    path_answer = node_rpc_server.rqmovesinit(rq_moves_node_id)
    verify_path_answer(path_answer)

    approach_position_joints = get_inverse_kin(approach_pose, qnear=approach_joints)
    movej(approach_position_joints)

    node_rpc_server.movejdefinewaypoint(rq_movej_node_id, get_actual_joint_positions(), 1.0, 1.0)
    node_rpc_server.setparentid(rq_movej_node_id, move_force_node_id)
    reset_node_executor()
    active_and_reset_node(move_force_node_id)
    node_execution_thread = execute_node(rq_movej_node_id, True)

    path_answer = node_rpc_server.rqmovesinit(rq_moves_node_id)
    verify_path_answer(path_answer)
    q0 = node_rpc_server.rqmovesgetfirstpoint(rq_moves_node_id)
    node_rpc_server.setparentid(rq_movej_node_id, move_force_node_id)
    node_rpc_server.movejdefinewaypoint(rq_movej_node_id, q0, 1.0, 0.4)
    execute_node(rq_movej_node_id)
    execute_node(start_waypoint_node_id)
    execute_node(end_waypoint_node_id)

    kill_thread(node_execution_thread)

    node_rpc_server.movejdefinewaypoint(rq_movej_node_id, get_actual_joint_positions(), 1.0, 1.0)
    node_rpc_server.setparentid(rq_movej_node_id, contact_force_node_id)
    reset_node_executor()
    active_and_reset_node(contact_force_node_id)
    node_execution_thread = execute_node(rq_movej_node_id, True)

    timeout = 20
    while (point_dist(get_actual_tcp_pose(), stop_pose) > end_reached_threshold):
      if (timeout <= 0):
        popup("Door has not reached its final position")
        halt
      else:
        sync()
        timeout = timeout - get_steptime()
      end
    end

    kill_thread(node_execution_thread)

    approach_pose_in_start_frame = pose_trans(pose_inv(start_pose), approach_pose)
    retract_pose = pose_trans(get_actual_tcp_pose(), approach_pose_in_start_frame)
    movej(retract_pose)

    node_rpc_server.deletenode(move_force_node_id)
    node_rpc_server.deletenode(rq_moves_node_id)
    node_rpc_server.deletenode(start_waypoint_node_id)
    node_rpc_server.deletenode(end_waypoint_node_id)
    node_rpc_server.deletenode(contact_force_node_id)
    node_rpc_server.deletenode(rq_movej_node_id)

  end

  ###################################################################################
  #
  # CNC Insertion
  #
  ###################################################################################

  def rq_collet_insertion(contact_pose, insert_pose, inserted_pose):
      movel(contact_pose, a=1.2, v=0.025)
      movel(insert_pose, a=1.2, v=0.025)

      rq_ft_sensor_disconnected_check()
      rq_zero_sensor()
      sleep(0.1)

      direction = "Z+"
      stop_force_threshold = 3.0
      max_radius = 5.0
      radius_incr = 0.7
      peck_mode = False
      tangential_speed = 0.02
      compliant_insert_force_threshold = 10.0
      spiral_initial_pose_offset_name = "spiral_initial_pose_offset_name"
      rq_ins_destination = inserted_pose
      max_distance = point_dist(inserted_pose, get_actual_tcp_pose())
      rq_spiral_not_completed = False
      rq_ins_speed_setting = 0.02

      rq_insert_spiral_urcap(direction, stop_force_threshold, max_radius, radius_incr, peck_mode, tangential_speed, compliant_insert_force_threshold, spiral_initial_pose_offset_name)

      if (rq_spiral_not_completed):
        return False
      end

      return True
  end

  def rq_push_part(approach_pose, chuck_pose):
      rq_ft_sensor_disconnected_check()
      rq_zero_sensor()
      sleep(0.1)

      # Find pose with z axis pointing in the direction of the insertion
      p1 = translate_to_origin(approach_pose)
      insertion_dir_in_base_frame = pose_trans(p1, pose_trans(pose_inv(approach_pose), chuck_pose))
      ref_frame_pose = list_to_pose(kinematics_rpc_server.poseFromZaxis([insertion_dir_in_base_frame[0], insertion_dir_in_base_frame[1], insertion_dir_in_base_frame[2]]))

      surface_found = rq_linear_search_custom_frame("Z+", 10.0, 0.025, 0.1, ref_frame_pose)

      if not(surface_found):
          return False
      end

      return True
  end

  def rq_place_in_chuck(close_chuck_do, open_chuck_do, chuck_approach, chuck_position, chuck_delay):
      rq_open_workholding(close_chuck_do, open_chuck_do)

      movel(chuck_approach, a=1.2, v=0.25)
      movel(chuck_position, a=1.2, v=0.25)

      rq_close_workholding(close_chuck_do, open_chuck_do)
      sleep(chuck_delay)
  end

  def rq_pre_pick_in_chuck(chuck_approach, chuck_position, speed=0.25, accel=1.2):
      movel(chuck_approach, accel, speed)
      movel(chuck_position, accel, speed)
  end

  def rq_post_pick_in_chuck(close_chuck_do, open_chuck_do, chuck_approach, chuck_position, chuck_delay, speed=0.25,
  accel=1.2):
      rq_open_workholding(close_chuck_do, open_chuck_do)
      sleep(chuck_delay)

      movel(chuck_approach, accel, speed)
  end

  def rq_open_workholding(close_do, open_do):
      rq_set_workholding_do(close_do, open_do, False)
  end

  def rq_close_workholding(close_do, open_do):
      rq_set_workholding_do(close_do, open_do, True)
  end

  def rq_set_workholding_do(close_do, open_do, close_request):
      is_close_do_valid = rq_is_do_valid(close_do)
      is_open_do_valid = rq_is_do_valid(open_do)

      if(is_close_do_valid):
          set_standard_digital_out(close_do, close_request)
      end
      if(is_open_do_valid):
          set_standard_digital_out(open_do, not close_request)
      end
      if(is_close_do_valid or is_open_do_valid):
          sleep(0.5)
      end
  end

  def rq_is_do_valid(do_id):
      return do_id >= 0 and do_id <= 7
  end

  def set_cleaning_digital_output(address, state, blow_off_mode, output_type):
     if(blow_off_mode == BLOW_OFF_MODE_SMART_AIR):
       rq_set_output(output_type, address, state)
     end
  end

  ###################################################################################
  #
  # PATH GENERATOR 6 POINTS CURVE BUILT WITH 2 POINTS
  #
  ###################################################################################

  def execute_half_pipe(pose_1, pose_2,pose_transformation_air_nozzle_to_actual_tcp, depth, length_distance, width, angle, speed, spacing, address, output_type, blow_off_mode, passes):
    path_gen_poses = get_path_generator_6_points_poses(pose_1, pose_2, pose_transformation_air_nozzle_to_actual_tcp, depth, length_distance, width, angle)
    start_pose = p[path_gen_poses[0,0],path_gen_poses[0,1],path_gen_poses[0,2],path_gen_poses[0,3],path_gen_poses[0,4],path_gen_poses[0,5]]
    path_generator_node_id = setup_path_generator_6_points(path_gen_poses, speed, spacing)
    execute_path_generator_6_points(path_generator_node_id, start_pose,  address, output_type, blow_off_mode, passes)
  end

  def get_path_generator_6_points_poses(pose_2, pose_5,pose_transformation_air_nozzle_to_actual_tcp, depth=0.01, length=0, width=0.05, angle_deg=0):

    def offset_pose(pose, offset, offset_reference_frame, pose_transformation_air_nozzle_to_actual_tcp):
      pose_relative_to_ref_frame = express_pose_A_relative_to_pose_B(pose, offset_reference_frame)
      ref_frame_with_offset = pose_trans(offset_reference_frame, offset)
      pose_with_offset = pose_trans(ref_frame_with_offset, pose_relative_to_ref_frame)
      pose_with_offset_for_actual_tcp = pose_trans(pose_with_offset, pose_transformation_air_nozzle_to_actual_tcp)
      return pose_to_list(pose_with_offset_for_actual_tcp)
    end

    if(length > 0):
      middle_pose = interpolate_pose(pose_2, pose_5, 0.5)

      poses = get_symmetric_poses_from_middle(pose_2, pose_5, middle_pose, length)
      pose_2 = poses[0]
      pose_5 = poses[1]
    end

    path_ref_frame = list_to_pose(kinematics_rpc_server.reorientP1WithXTowardP2andZApproxP1Z(pose_2, pose_5))

    offset1 = pose_add(p[0,0,0,0,d2r(angle_deg),0], p[0, width,-depth,-d2r(angle_deg),0,0])
    offset2 = pose_add(p[0,0,0,0,d2r(angle_deg),0], p[0,     0,     0,              0,0,0])
    offset3 = pose_add(p[0,0,0,0,d2r(angle_deg),0], p[0,-width,-depth, d2r(angle_deg),0,0])

    pose_1_array = offset_pose(pose_2, offset1, path_ref_frame, pose_transformation_air_nozzle_to_actual_tcp)
    pose_2_array = offset_pose(pose_2, offset2, path_ref_frame, pose_transformation_air_nozzle_to_actual_tcp)
    pose_3_array = offset_pose(pose_2, offset3, path_ref_frame, pose_transformation_air_nozzle_to_actual_tcp)

    pose_4_array = offset_pose(pose_5, offset1, path_ref_frame, pose_transformation_air_nozzle_to_actual_tcp)
    pose_5_array = offset_pose(pose_5, offset2, path_ref_frame, pose_transformation_air_nozzle_to_actual_tcp)
    pose_6_array = offset_pose(pose_5, offset3, path_ref_frame, pose_transformation_air_nozzle_to_actual_tcp)

    return [pose_1_array, pose_2_array, pose_3_array, pose_4_array, pose_5_array, pose_6_array]
  end

  def setup_path_generator_6_points(pose_list, tcp_speed=0.1, spacing=0.02):

    def json_path_generator_node(pose_list, tcp_speed, spacing):

      SIX_POINTS_CURVE = 3
      OFFSET_TYPE_NONE = 0
      FORCE_OPPOSITE_SIDE = 2

      json = "{"
      json = concat(json, key_val("tcpSpeed", tcp_speed), ",")
      json = concat(json, key_val("poses", pose_list), ",")
      json = concat(json, key_val("avoidAbruptEnd", "false"), ",")
      json = concat(json, key_val("isSurfaceFillOn", "true"), ",")
      json = concat(json, key_val("spacing", spacing), ",")
      json = concat(json, key_val("pathType", SIX_POINTS_CURVE), ",")
      json = concat(json, key_val("offsetType",OFFSET_TYPE_NONE), ",")
      json = concat(json, key_val("endingMode", FORCE_OPPOSITE_SIDE), "}")

      return json
    end

    rq_path_generator_parent_id = 0
    path_generator_node_id = node_rpc_server.createPathGeneratorNode()
    node_rpc_server.fromjson(path_generator_node_id, json_path_generator_node(pose_list, tcp_speed, spacing))
    node_rpc_server.setparentid(path_generator_node_id, rq_path_generator_parent_id)

    return path_generator_node_id
  end

  def execute_path_generator_6_points(path_generator_node_id, pose_1, address = INVALID_OUTPUT_ADDRESS, output_type = MODBUS_TYPE, blow_off_mode = BLOW_OFF_MODE_NO_AIR, passes = 1):
    index = 0
    while (index < passes):
      movej(get_inverse_kin(pose_1))
      set_cleaning_digital_output(address, True, blow_off_mode, output_type)
      reset_node_executor()
      node_execution_thread = execute_node(path_generator_node_id, True)
      rq_continue_node_execution = False
      set_cleaning_digital_output(address, False, blow_off_mode, output_type)
      join node_execution_thread
      index = index + 1
    end
    node_rpc_server.deletenode(path_generator_node_id)
  end

  ###################################################################################
  #
  # Straight line trajectory
  #
  ###################################################################################

  def execute_straight_line(p1, p2,pose_transformation_air_nozzle_to_actual_tcp, accel=1.2, speed=0.25, distance = 0, angles = [0, 0, 0], address = INVALID_OUTPUT_ADDRESS, output_type = MODBUS_TYPE, blow_off_mode = BLOW_OFF_MODE_NO_AIR, passes = 1):
    offset_for_angles = p[0, 0, 0, d2r(angles[0]), d2r(angles[1]), d2r(angles[2])]
    p1 = pose_trans(p1, offset_for_angles)
    p2 = pose_trans(p2, offset_for_angles)

    # apply transformation to take into account that the actual tcp offset is not the same as the one that was used when the waypoints were saved:
    p1 = pose_trans(p1, pose_transformation_air_nozzle_to_actual_tcp)
    p2 = pose_trans(p2, pose_transformation_air_nozzle_to_actual_tcp)
    global air_output_adress = address

    qActual = get_actual_joint_positions()
    CleanPathId = node_rpc_server.createnewcleaningpathnode(p1, p2, qActual, passes, distance, accel, speed, blow_off_mode)

    reset_node_executor()
    if output_type == MODBUS_TYPE:
      air_thread = run modbusAirControlThread()
    elif output_type == STANDARD_TYPE:
      air_thread = run standardAirControlThread()
    end

    node_execution_thread = execute_node(CleanPathId, True)
    rq_continue_node_execution = False

    join node_execution_thread
    node_rpc_server.deletenode(CleanPathId)
    if output_type == MODBUS_TYPE or output_type == STANDARD_TYPE :
      kill air_thread
    end
  end

  ###################################################################################
  #
  # Cross trajectory
  #
  ###################################################################################

  def find_cross_trajectory_poses(p1, p2, height=0, width=0, p1_angles = [0, 0, 0], p2_angles = [0, 0, 0], p3_angles = [0, 0, 0], p4_angles = [0, 0, 0]):
    def find_side_poses(p0, p1):
      def find_side_pose(p0,p1,angle):
        p1_T_p0 = pose_trans(pose_inv(p0), p1)
        rotated_p0_by_90_degrees = pose_trans(p0, p[0, 0, 0, 0, 0, d2r(angle)])

        side_pose = pose_trans(rotated_p0_by_90_degrees, p1_T_p0)
        side_pose[3] = p0[3]
        side_pose[4] = p0[4]
        side_pose[5] = p0[5]

        return side_pose
      end

      p3= find_side_pose(p0, p1, 90)
      p4 = find_side_pose(p0, p1, 270)

      return [p3, p4]
    end

    def get_start_and_end_poses_based_on_distance(p1, p2, middle_pose, distance):
      if(distance == 0):
        start_pose = p1
        end_pose = p2
      else:
        poses = get_symmetric_poses_from_middle(p1, p2, middle_pose, distance)
        start_pose = poses[0]
        end_pose = poses[1]
      end
      return [start_pose, end_pose]
    end

    def get_side_poses_based_on_distance(p1, p2, middle_pose, width):
      if(width == 0):
        side_poses = find_side_poses(middle_pose, p1)
      else:
        poses = get_symmetric_poses_from_middle(p1, p2, middle_pose, width)
        side_poses = find_side_poses(middle_pose, poses[0])
      end

      return side_poses
    end

    def get_angle_offset(angles):
      return  p[0, 0, 0, d2r(angles[0]), d2r(angles[1]), d2r(angles[2])]
    end

    middle_pose = interpolate_pose(p1, p2, 0.5)

    start_and_end_poses = get_start_and_end_poses_based_on_distance(p1, p2, middle_pose, height)
    side_poses = get_side_poses_based_on_distance(p1, p2, middle_pose, width)

    p1_offset = get_angle_offset(p1_angles)
    p2_offset = get_angle_offset(p2_angles)
    p3_offset = get_angle_offset(p3_angles)
    p4_offset = get_angle_offset(p4_angles)

    start_and_end_poses[0] = pose_trans(start_and_end_poses[0], p1_offset)
    start_and_end_poses[1] = pose_trans(start_and_end_poses[1], p2_offset)
    side_poses[0] = pose_trans(side_poses[0], p3_offset)
    side_poses[1] = pose_trans(side_poses[1], p4_offset)

    return [middle_pose, start_and_end_poses[0], start_and_end_poses[1], side_poses[0], side_poses[1]]
  end

  def execute_cross_trajectory(p1, p2,pose_transformation_air_nozzle_to_actual_tcp, height=0, width=0, p1_angles = [0, 0, 0], p2_angles = [0, 0, 0], p3_angles = [0, 0, 0], p4_angles = [0, 0, 0], accel=1.2, speed=0.25,  address = INVALID_OUTPUT_ADDRESS, output_type = MODBUS_TYPE, blow_off_mode = BLOW_OFF_MODE_NO_AIR, passes = 1):

    cross_poses = find_cross_trajectory_poses(p1, p2, height, width, p1_angles, p2_angles, p3_angles, p4_angles)

    p0 = pose_trans(cross_poses[0], pose_transformation_air_nozzle_to_actual_tcp)
    p1 = pose_trans(cross_poses[1], pose_transformation_air_nozzle_to_actual_tcp)
    p2 = pose_trans(cross_poses[2], pose_transformation_air_nozzle_to_actual_tcp)
    p3 = pose_trans(cross_poses[3], pose_transformation_air_nozzle_to_actual_tcp)
    p4 = pose_trans(cross_poses[4], pose_transformation_air_nozzle_to_actual_tcp)

   index = 0

   while (index < passes):
     movej(get_inverse_kin(p0))
     set_cleaning_digital_output(address, True, blow_off_mode, output_type)
     movel(p1, accel, speed)
     movel(p2, accel, speed)
     movel(p0, accel, speed)
     movel(p3, accel, speed)
     movel(p4, accel, speed)
     set_cleaning_digital_output(address, False, blow_off_mode, output_type)
     index = index + 1
   end
  end

  def execute_waypoint_cross_trajectory(starting_pose, finishing_pose, accel=1.2, speed=0.25):
   movej(get_inverse_kin(starting_pose))
   movel(finishing_pose, accel, speed)
  end

  ###################################################################################
  #
  # Fermat spiral trajectory
  #
  ###################################################################################

  def execute_fermat_spiral(start_pose, end_pose,pose_transformation_air_nozzle_to_actual_tcp, max_radius = 0, angle = 0, number_of_turns = 1, speed = 0.25,address = INVALID_OUTPUT_ADDRESS, output_type = MODBUS_TYPE, blow_off_mode = BLOW_OFF_MODE_NO_AIR, passes = 1):
    def find_middle(start_pose, end_pose):
      alpha = 0.5
      return interpolate_pose(start_pose, end_pose, alpha)
    end

    def find_next_theta(spiral_constant, theta, speed):
      denom = spiral_constant * sqrt(1/(4*theta) + theta)
      theta_dot = speed / denom
      theta = theta + theta_dot * rq_controller_time_step
      return theta
    end

    def find_spiral_pose(theta, spiral_plane, center_pose, angle, spiral_constant, pose_transformation_air_nozzle_to_actual_tcp):
      local r = spiral_constant * sqrt(theta)
      local x = r * cos(theta)
      local y = r * sin(theta)

      local p2 = pose_trans(spiral_plane, p[x,y,0,0,0,0])
      local p3 = p[p2[0], p2[1], p2[2], center_pose[3], center_pose[4], center_pose[5]]
      local p4 = pose_trans(p3, pose_transformation_air_nozzle_to_actual_tcp)
      local p5 = pose_trans(p4, p[0, 0, 0, -d2r(angle)*cos(theta), -d2r(angle)*sin(theta), 0])
      return p5
    end

    def execute_outer_to_inner_spiral(start_pose, middle_pose, spiral_plane, pose_transformation_air_nozzle_to_actual_tcp, max_angle, angle, spiral_constant_nominal, speed, address, output_type, blow_off_mode):
      local theta = max_angle
      local max_r = point_dist(start_pose, middle_pose)
      local spiral_constant = -1 * spiral_constant_nominal
      local r = max_r
      local is_first_pose = True

      while (norm((r)) <= max_r):
        theta = find_next_theta(spiral_constant, theta, speed)
        if(theta < 0):
          break
        end

        r = spiral_constant * sqrt(theta)
        next_pose = find_spiral_pose(theta, spiral_plane, middle_pose, angle, spiral_constant, pose_transformation_air_nozzle_to_actual_tcp)

        if (is_first_pose):
          movej(get_inverse_kin(next_pose))
          set_cleaning_digital_output(address, True, blow_off_mode, output_type)
          is_first_pose = False
        else:
          servoj(get_inverse_kin(next_pose), t = rq_controller_time_step)
        end
      end
    end

    def execute_inner_to_outer_spiral(start_pose, middle_pose, spiral_plane, pose_transformation_air_nozzle_to_actual_tcp, angle, spiral_constant, speed):
      local theta = 0.0001
      local max_r = point_dist(start_pose, middle_pose)
      local r = 0

      while (norm(r) <= max_r):
        theta = find_next_theta(spiral_constant, theta, speed)
        r = spiral_constant * sqrt(theta)
        next_pose = find_spiral_pose(theta, spiral_plane, middle_pose, angle, spiral_constant, pose_transformation_air_nozzle_to_actual_tcp)
        servoj(get_inverse_kin(next_pose), t = rq_controller_time_step)
      end
    end

    max_angle = d2r(number_of_turns * 360)
    middle_pose = find_middle(start_pose, end_pose)

    if(max_radius > 0):
      poses = get_symmetric_poses_from_middle(start_pose, end_pose, middle_pose, max_radius * 2)
      start_pose = poses[0]
      end_pose = poses[1]
    end

    SPIRAL_CONSTANT = (point_dist(middle_pose, start_pose)) / sqrt(max_angle)

    spiral_plane = list_to_pose(kinematics_rpc_server.reorientP1WithXTowardP2andZApproxP1Z(middle_pose, end_pose))


    index = 0
    while(index < passes):
      execute_outer_to_inner_spiral(start_pose, middle_pose, spiral_plane,pose_transformation_air_nozzle_to_actual_tcp, max_angle, angle, SPIRAL_CONSTANT, speed, address, output_type, blow_off_mode)
      execute_inner_to_outer_spiral(end_pose, middle_pose, spiral_plane, pose_transformation_air_nozzle_to_actual_tcp, angle, SPIRAL_CONSTANT, speed)
      set_cleaning_digital_output(address, False, blow_off_mode, output_type)
      index = index + 1
    end
  end

  ###################################################################################
  #
  # ROBOTIQ VISE INSERTION
  #
  # - The first touch is performed in the direction of the gravity, regardless of
  #   the robot mounting orientation, tcp offset and TCP orientation
  # - Optional 2e et 3e touch are performed relative to TCP. They require that, at
  #   the moment that the insertion is performed, the TCP is oriented such that one
  #   axis is aligned with the gravity. The TCP axes for the 2e and 3e touch are
  #   chosen as the ones not aligned with the gravity.
  ###################################################################################
  def insert_in_vise(start_pose, end_pose, number_of_touch=3, forces=[10, 20, 20], invert_axis=False, move_to_end_pose=False):

    def list_by_scalar_multiply_(l1, scalar):
      result = l1
      i=0
      while i<length(result):
        result[i]=l1[i]*scalar
        i=i+1
      end
      return result
    end

    def find_gravity_direction(acceleration_direction, threshold):
      result = [False, False, False]
      i = 0
      while i < length(result):
        result[i] =  norm(acceleration_direction[i]) > threshold
        i = i + 1
      end
      return result
    end

    def get_axis(index, direction):
      axis = "XYZ"
      if direction < 0:
        sign = "-"
      elif direction > 0:
        sign = "+"
      else:
        popup("insert_in_vise:get_axis >>> direction cannot be 0. Fix it.")
        halt
      end
      return str_cat(str_sub(axis, index, 1), sign)
    end

    def direction_to_index(str):
      if "X" == str_sub(str, 0, 1):
        return 0
      elif "Y" == str_sub(str, 0, 1):
        return 1
      elif "Z" == str_sub(str, 0, 1):
        return 2
      else:
        popup("invalid direction :", str)
        halt
      end
    end

    def find_touch_direction(mask, direction):
      i = 0
      result = [0, 0, 0]
      while i < 3:
        if mask[i]:
          result[i] = direction[i]
        end
        i = i + 1
      end
      return result
    end

    def find_touch_direction_str(mask, direction):
      i = 0
      result = ""
      while i < 3:
        if mask[i]:
          result = str_cat(result, get_axis(i, direction[i]))
        end
        i = i + 1
      end
      return result
    end

    def invert(list):
      result = list
      i = 0
      while i < length(list):
        result[i] = not list[i]
        i = i + 1
      end
      return result
    end

    def assert_that_the_first_touch_is_aligned_with_an_axis(first_touch_direction_mask):
      i = 0
      counter = 0
      while i < length(first_touch_direction_mask):
        if first_touch_direction_mask[i]:
          counter = counter + 1
        end
        i = i + 1
      end

      if counter != 1:
        popup("One of the TCP axes must be perpendicular to the floor while loading the part in the vise.")
        halt
      end
    end

    def setup_nodes(forces, number_of_touch, first_touch_direction_mask, direction, second_direction_str, third_direction_str):
      def max_deviation_from(forces, enabled_axis):
        i = 0
        deviation = [0, 0, 0, 0, 0, 0]
        while i < 3:
          if forces[i] > 0:
            deviation[i] = 10
          elif forces[i] ==  0:
            deviation[i] = 10
          end
          i = i + 1
        end
        while i < 6:
          if enabled_axis[i]:
            deviation[i] = 0.35
          end
          i = i + 1
        end
        return deviation
      end

      def min_deviation_from(forces, enabled_axis):
        i = 0
        deviation = [0, 0, 0, 0, 0, 0]
        while i < 3:
          if forces[i] < 0:
            deviation[i] = -10
          elif forces[i] ==  0:
            deviation[i] = -10
          end
          i = i + 1
        end
        while i < 6:
          if enabled_axis[i]:
            deviation[i] = -0.35
          end
          i = i + 1
        end
        return deviation
      end

      def stiffness_from(forces):
        i = 0
        stiffness = [0, 0, 0, 100, 100, 100]
        while i < length(forces):
          if norm(forces[i]) > 0:
            stiffness[i] = 100
          else:
            stiffness[i] = 85
          end
          i = i + 1
        end
        return stiffness
      end

      def compute_final_forces(forces, number_of_touch, first_touch_direction_mask, direction, second_direction_str, third_direction_str):
        final_forces = [0, 0, 0]
        if number_of_touch > 0:
          i = 0
          while i < length(first_touch_direction_mask):
            if first_touch_direction_mask[i]:
              break
            end
            i = i + 1
          end
          final_forces[i] = direction[i] * forces[i]
        end
        if number_of_touch > 1:
          i = direction_to_index(second_direction_str)
          final_forces[i] = direction[i] * forces[i]
        end
        if number_of_touch > 2:
          i = direction_to_index(third_direction_str)
          final_forces[i] = direction[i] * forces[i]
        end
        return final_forces
      end

      def compute_enabled_axis(first_touch_direction_mask):
        enabled_axis = [True, True, True, False, False, False]
        i = 0
        while i < length(first_touch_direction_mask):
          if first_touch_direction_mask[i]:
            break
          end
          i = i + 1
        end
        enabled_axis[i + 3] = True

        return enabled_axis
      end

      final_forces = compute_final_forces(forces, number_of_touch, first_touch_direction_mask, direction, second_direction_str, third_direction_str)
      enabled_axis = compute_enabled_axis(first_touch_direction_mask)

      force_node_id = rq_setup_machine_tending_force_node(1, [final_forces[0], final_forces[1], final_forces[2], 0, 0, 0], stiffness_from
      (final_forces), min_deviation_from(final_forces, enabled_axis), max_deviation_from(final_forces, enabled_axis), rq_bool_array_to_string(enabled_axis), "false")
      movej_node_id = node_rpc_server.createnewmovejnode()
      node_rpc_server.setparentid(movej_node_id, force_node_id)

      return [force_node_id, movej_node_id]
    end

    def average_tool_acceleration_reading(n_samples, delay):
      n = n_samples
      reading = [0, 0, 0]
      while n > 0:
        reading = reading + get_tool_accelerometer_reading()
        sleep(delay)
        n = n - 1
      end
      return reading/n_samples
    end

    def linear_search_toward_gravity(force):
      # maybe add a stopj here to prevent acceleration reading to be influenced by robot movement
      flange_accel = average_tool_acceleration_reading(10, 0.1) # measured accel is oriented in gravity oposite direction
      flange_accel_pose = p[-flange_accel[0], -flange_accel[1], -flange_accel[2], 0, 0,0]
      p1 = translate_to_origin(get_actual_tool_flange_pose())
      gravity_dir_in_base_frame = pose_trans(p1, flange_accel_pose)

      # Find pose with z axis pointing in gravity direction:
      ref_frame_pose = list_to_pose(kinematics_rpc_server.poseFromZaxis([gravity_dir_in_base_frame[0], gravity_dir_in_base_frame[1], gravity_dir_in_base_frame[2]]))
      speed = 0.01
      abs_max_distance = 0.05

      surface_found = rq_linear_search_custom_frame("Z+", force, speed, abs_max_distance, ref_frame_pose)
      return surface_found
    end

    #### Actual insert_in_vise method ####
    movel(start_pose)
    zero_ftsensor()

    # 1. Use accelerometer reading to find touches directions:
    ACCELERATION_THRESHOLD = 8
    flange_accel = average_tool_acceleration_reading(10, 0.1)
    tcp_accel = pose_trans(pose_inv(get_tcp_offset()), p[flange_accel[0], flange_accel[1], flange_accel[2], 0, 0, 0])
    first_touch_direction_mask = find_gravity_direction(tcp_accel, ACCELERATION_THRESHOLD)
    assert_that_the_first_touch_is_aligned_with_an_axis(first_touch_direction_mask)

    direction_transform = pose_trans(pose_inv(start_pose), end_pose)
    direction = [direction_transform[0], direction_transform[1], direction_transform[2]]
    direction_sign = [direction[0]/norm(direction[0]), direction[1]/norm(direction[1]), direction[2]/norm(direction[2])]

    touch_direction_str = find_touch_direction_str(invert(first_touch_direction_mask), direction_sign)
    touch_direction = find_touch_direction(invert(first_touch_direction_mask), direction_sign)

    if invert_axis:
      second_direction_str = str_sub(touch_direction_str, 0, 2)
      third_direction_str = str_sub(touch_direction_str, 2, 4)
    else:
      second_direction_str = str_sub(touch_direction_str, 2, 4)
      third_direction_str = str_sub(touch_direction_str, 0, 2)
    end

    end_pose_orientation = translate_to_origin(end_pose)

    # 2. Prepare nodes:
    rq_cnc_insertion_node_ids = setup_nodes(forces, number_of_touch, first_touch_direction_mask, direction_sign, second_direction_str, third_direction_str)
    feature_tool = 1

    # 3. Perform touches:
    if number_of_touch > 0:
      surface_found = linear_search_toward_gravity(forces[0])
      if not surface_found:
        textmsg("Insertion in vise: First contact has not been found")
        popup("First contact has not been found", title="Insertion in vise", blocking=True)
        return UNDEFINED_THREAD_ID
      end
    end
    if number_of_touch > 1:
      surface_found = rq_linear_search_urcap(second_direction_str, forces[1], 0.01, 0.05, feature_tool)
      if not surface_found:
        textmsg("Insertion in vise: Second contact has not been found")
        popup("Second contact has not been found", title="Insertion in vise", blocking=True)
        return UNDEFINED_THREAD_ID
      end
    end
    if number_of_touch > 2:
      surface_found = rq_linear_search_urcap(third_direction_str, forces[2], 0.01, 0.05, feature_tool)
      if not surface_found:
        textmsg("Insertion in vise: Third contact has not been found")
        popup("Third contact has not been found", title="Insertion in vise", blocking=True)
        return UNDEFINED_THREAD_ID
      end
    end

    # 4. Move to end position:
    if not move_to_end_pose:
      end_pose = get_actual_tcp_pose()
    end

    node_rpc_server.movejdefinewaypoint(rq_cnc_insertion_node_ids[1], get_actual_joint_positions(), 1.0, 1.0)
    reset_node_executor()
    active_and_reset_node(rq_cnc_insertion_node_ids[0])
    node_execution_thread = execute_node(rq_cnc_insertion_node_ids[1], True)
    node_rpc_server.movejdefinewaypoint(rq_cnc_insertion_node_ids[1], get_inverse_kin(end_pose), 1.0, 1.0)
    execute_node(rq_cnc_insertion_node_ids[1])
    sleep(1)
    return node_execution_thread
  end

  ###################################################################################
  # AIR OUTPUT CONTROL
  ###################################################################################
  thread modbusAirControlThread():
    while (True):
      rq_air_value = read_input_boolean_register(101)
      modbus_set_output_signal(air_output_adress, rq_air_value, False)
      sleep(rq_controller_time_step)
    end
  end

  thread standardAirControlThread():
    while (True):
      rq_air_value = read_input_boolean_register(101)
      set_digital_out(air_output_adress, rq_air_value)
      sleep(rq_controller_time_step)
    end
  end
  def rq_set_output(output_type, address, value):
    if output_type == "MODBUS":
      modbus_set_output_signal(address, value)
    elif output_type == "STANDARD":
      set_standard_digital_out(address, value)
    end
  end

  def rq_digital_output_action(action, output_type, address, time_on=1, time_off=0.5, delay_after=0):
    if action == "PUSH_AND_HOLD":
      rq_set_output(output_type, address, True)
    elif action == "PUSH":
      rq_set_output(output_type, address, True)
      sleep(time_on)
      rq_set_output(output_type, address, False)
    elif action == "DOUBLE_PUSH":
      rq_set_output(output_type, address, True)
      sleep(time_on)
      rq_set_output(output_type, address, False)
      sleep(time_off)
      rq_set_output(output_type, address, True)
      sleep(time_on)
      rq_set_output(output_type, address, False)
    elif action == "RELEASE":
      rq_set_output(output_type, address, False)
    end
    sleep(delay_after)
  end
  def json_kinematic_parameters_ratio(ratio):
    json = "{"
    json = concat(json, key_val("kinematicParametersRatio", ratio), "}")
    return json
  end

  def execute_move_along_trail(trail_node_id, joint_positions, kinematic_parameters_ratio):
    node_rpc_server.fromjson(trail_node_id, json_kinematic_parameters_ratio(kinematic_parameters_ratio))
    roadmap_state = node_rpc_server.initRoadmap(trail_node_id, joint_positions)
    path_time = roadmap_state[0]

    if(path_time > 0.0):
      reset_node_executor()
      node_execution_thread = execute_node(trail_node_id, True)
      kill node_execution_thread
    end
  end
    global servojId = 2
  rq_collision_detection_start(60.0,10.0, False)
  # end: URCap Installation Node
  while (True):
    $ 1 "Robot Program"
    # begin: URCap Program Node
    #   Source: Robotiq_3-Finger_Adaptive_Gripper, 1.0.1, Robotiq inc.
    #   Type: 3F Gripper Move
    $ 2 "3F Pinch Open"
    rq_set_pinch()
    rq_set_force(255)
    rq_set_speed(255)
    rq_move_wait(80)
    # end: URCap Program Node
  end
end_1222
